Staubli VAL3: external.pjx

--- external.pjx ---
Parameters version=s7.9.4 stackSize=5000 millimeterUnit=true
Program file=aLight1.pgx
Program file=aLight2.pgx
Program file=aLight3.pgx
Program file=iCryoLongIn.pgx
Program file=iCryoShortIn.pgx
Program file=iEmergencyIn.pgx
Program file=iFluor.pgx
Program file=iFluorClosed.pgx
Program file=iFluorOpen.pgx
Program file=iGrip.pgx
Program file=iGripClosed.pgx
Program file=iGripOpen.pgx
Program file=iHeater.pgx
Program file=iIdent1.pgx
Program file=iIdent2.pgx
Program file=iIdent3.pgx
Program file=iLevel1.pgx
Program file=iLevel2.pgx
Program file=iLevel3.pgx
Program file=iLevel4.pgx
Program file=iLevel5.pgx
Program file=iLevelFault.pgx
Program file=iLidClosed.pgx
Program file=iPilatusPos.pgx
Program file=iPlate1.pgx
Program file=iPlate2.pgx
Program file=iPlate3.pgx
Program file=iPressureSensor.pgx
Program file=iRack1.pgx
Program file=iRack2.pgx
Program file=iRack3.pgx
Program file=iRack4.pgx
Program file=iSample.pgx
Program file=iSchock.pgx
Program file=iState.pgx
Program file=iTeste.pgx
Program file=iTool.pgx
Program file=ioLinks.pgx
Program file=oCryoLongOut.pgx
Program file=oCryoShortOut.pgx
Program file=oEmergencyOut.pgx
Program file=oFluorDet.pgx
Program file=oGripCmd.pgx
Program file=oGripCmd2.pgx
Program file=oHeater.pgx
Program file=oHeaterTask.pgx
Program file=oLid.pgx
Program file=oPilatusCover.pgx
Program file=oResetFault.pgx
Program file=oSample.pgx
Program file=oShutter.pgx
Program file=oVacuumValve.pgx
Program file=power.pgx
Program file=start.pgx
Program file=stop.pgx
Data file=external.dtx
Library alias=io path=io autoload=true password=

--- external.dtx ---
public aio aHeaterTime[2]
public aio aLight1[2]
public aio aLight2[2]
public aio aLight3[2]
public aio aState
public dio iCryoLongIn
public dio iCryoShortIn
public dio iEmergencyIn
public dio iFluor
public dio iFluorClosed
public dio iFluorOpen
public dio iGrip
public dio iGripClosed
public dio iGripOpen
public dio iHeaterStatus
public dio iIdent1
public dio iIdent2
public dio iIdent3
public dio iLevel1
public dio iLevel2
public dio iLevel3
public dio iLevel4
public dio iLevel5
public dio iLevelFault
public dio iLidClosed
public dio iPilatusPos
public dio iPlate1
public dio iPlate2
public dio iPlate3
public dio iPressureSensor
public dio iRack1
public dio iRack2
public dio iRack3
public dio iRack4
public dio iSampleStatus
public dio iSchock
public dio iTeste
public dio iTool
public dio oCryoLongOut
public dio oCryoShortOut
public dio oEmergencyOut
public dio oFluorDet
public dio oGripCmd
public dio oGripCmd2
public dio oHeater
public dio oLid
public dio oPilatusCover
public dio oResetFault
public dio oSample
public dio oShutter
public dio oVacuumValve
public mdesc mNomSpeed = {blend=off}

--- start.pgx ---
public program start()
begin
  call ioLinks()
end

--- aLight1.pgx ---
public program aLight1(num nValue (dimensions=1))
begin
  aioSet(aLight1,nValue)
end

--- aLight2.pgx ---
public program aLight2(num nValue (dimensions=1))
begin
  aioSet(aLight2,nValue)
end

--- aLight3.pgx ---
public program aLight3(num nValue (dimensions=1))
begin
  aioSet(aLight3,nValue)
end

--- iCryoLongIn.pgx ---
public program iCryoLongIn(num& nNum[] (dimensions=1))
begin
  nNum=dioGet(iCryoLongIn)
end

--- iCryoShortIn.pgx ---
public program iCryoShortIn(num& nNum[] (dimensions=1))
begin
  nNum=dioGet(iCryoShortIn)
end

--- iEmergencyIn.pgx ---
public program iEmergencyIn(num& nNum[] (dimensions=1))
begin
  nNum=dioGet(iEmergencyIn)
end

--- iFluor.pgx ---
public program iFluor(num& nNum[] (dimensions=1))
begin
  if (dioGet(iFluorClosed)==0) and (dioGet(iFluorOpen)==1)
    nNum=1
  endIf
  if (dioGet(iFluorClosed)==1) and (dioGet(iFluorOpen)==0)
    nNum=0
  endIf
end

--- iFluorClosed.pgx ---
public program iFluorClosed(num& nNum[] (dimensions=1))
begin
  nNum=dioGet(iFluorClosed)
end

--- iFluorOpen.pgx ---
public program iFluorOpen(num& nNum[] (dimensions=1))
begin
  nNum=dioGet(iFluorOpen)
end

--- iGrip.pgx ---
public program iGrip(num& nNum[] (dimensions=1))
begin
  if (dioGet(iGripClosed)==0) and (dioGet(iGripOpen)==1)
    nNum=1
  endIf
  if (dioGet(iGripClosed)==1) and (dioGet(iGripOpen)==0)
    nNum=0
  endIf
end

--- iGripClosed.pgx ---
public program iGripClosed(num& nNum[] (dimensions=1))
begin
  nNum=dioGet(iGripClosed)
end

--- iGripOpen.pgx ---
public program iGripOpen(num& nNum[] (dimensions=1))
begin
  nNum=dioGet(iGripOpen)
end

--- iHeater.pgx ---
public program iHeater(num& nNum[] (dimensions=1))
begin
  nNum=dioGet(iHeaterStatus)
end

--- iIdent1.pgx ---
public program iIdent1(num& nNum[] (dimensions=1))
begin
  nNum=dioGet(iIdent1)
end

--- iIdent2.pgx ---
public program iIdent2(num& nNum[] (dimensions=1))
begin
  nNum=dioGet(iIdent2)
end

--- iIdent3.pgx ---
public program iIdent3(num& nNum[] (dimensions=1))
begin
  nNum=dioGet(iIdent3)
end

--- iLevel1.pgx ---
public program iLevel1(num& nNum[] (dimensions=1))
begin
  nNum=dioGet(iLevel1)
end

--- iLevel2.pgx ---
public program iLevel2(num& nNum[] (dimensions=1))
begin
  nNum=dioGet(iLevel2)
end

--- iLevel3.pgx ---
public program iLevel3(num& nNum[] (dimensions=1))
begin
  nNum=dioGet(iLevel3)
end

--- iLevel4.pgx ---
public program iLevel4(num& nNum[] (dimensions=1))
begin
  nNum=dioGet(iLevel4)
end

--- iLevel5.pgx ---
public program iLevel5(num& nNum[] (dimensions=1))
begin
  nNum=dioGet(iLevel5)
end

--- iLevelFault.pgx ---
public program iLevelFault(num& nNum[] (dimensions=1))
begin
  nNum=dioGet(iLevelFault)
end

--- iLidClosed.pgx ---
public program iLidClosed(num& nNum[] (dimensions=1))
begin
  nNum=dioGet(iLidClosed)
end

--- ioLinks.pgx ---
program ioLinks()
begin
  dioLink(iEmergencyIn,io:EmergencyIn)
  dioLink(iSchock,io:Schock)
  dioLink(iGripOpen,io:GripOpen)
  dioLink(iGripClosed,io:GripClosed)
  dioLink(iRack1,io:Rack1)
  dioLink(iRack2,io:Rack2)
  dioLink(iRack3,io:Rack3)
  dioLink(iRack4,io:Rack4)
  dioLink(iIdent1,io:Ident1)
  dioLink(iIdent2,io:Ident2)
  dioLink(iIdent3,io:Ident3)
  dioLink(iPressureSensor,io:PressureSensor)
  dioLink(iCryoShortIn,io:CryoShortIn)
  dioLink(iCryoLongIn,io:CryoLongIn)
  dioLink(iPilatusPos,io:PilatusPos)
  dioLink(iPlate1,io:Plate1)
  dioLink(iPlate2,io:Plate2)
  dioLink(iPlate3,io:Plate3)
  dioLink(iLevelFault,io:LevelFault)
  dioLink(iLevel1,io:Level1)
  dioLink(iLevel2,io:Level2)
  dioLink(iLevel3,io:Level3)
  dioLink(iLevel4,io:Level4)
  dioLink(iLevel5,io:Level5)
  dioLink(iLidClosed,io:LidClosed)
  dioLink(iFluorOpen,io:FluorOpen)
  dioLink(iFluorClosed,io:FluorClosed)
  dioLink(iHeaterStatus,io:HeaterStatus)
  dioLink(iSampleStatus,io:SampleStatus)
  dioLink(oResetFault,io:ResetFault)
  dioLink(oEmergencyOut,io:EmergencyOut)
  dioLink(oCryoShortOut,io:CryoShortOut)
  dioLink(oCryoLongOut,io:CryoLongOut)
  dioLink(oFluorDet,io:FluorDet)
  dioLink(oPilatusCover,io:PilatusCover)
  dioLink(oLid,io:Lid)
  dioLink(oHeater,io:Heater)
  dioLink(oShutter,io:Shutter)
  dioLink(oVacuumValve,io:VacuumValve)
  dioLink(oGripCmd,io:valve1)
  dioLink(oGripCmd2,io:valve2)
  dioLink(oSample,io:Sample)
  aioLink(aLight1,io:Light1)
  aioLink(aLight2,io:Light2)
  aioLink(aLight3,io:Light3)
  aioLink(aHeaterTime,io:HeaterTime)
end

--- iPilatusPos.pgx ---
public program iPilatusPos(num& nNum[] (dimensions=1))
begin
  nNum=dioGet(iPilatusPos)
end

--- iPlate1.pgx ---
public program iPlate1(num& nNum[] (dimensions=1))
begin
  nNum=dioGet(iPlate1)
end

--- iPlate2.pgx ---
public program iPlate2(num& nNum[] (dimensions=1))
begin
  nNum=dioGet(iPlate2)
end

--- iPlate3.pgx ---
public program iPlate3(num& nNum[] (dimensions=1))
begin
  nNum=dioGet(iPlate3)
end

--- iPressureSensor.pgx ---
public program iPressureSensor(num& nNum[] (dimensions=1))
begin
  nNum=dioGet(iPressureSensor)
end

--- iRack1.pgx ---
public program iRack1(num& nNum[] (dimensions=1))
begin
  nNum=dioGet(iRack1)
end

--- iRack2.pgx ---
public program iRack2(num& nNum[] (dimensions=1))
begin
  nNum=dioGet(iRack2)
end

--- iRack3.pgx ---
public program iRack3(num& nNum[] (dimensions=1))
begin
  nNum=dioGet(iRack3)
end

--- iRack4.pgx ---
public program iRack4(num& nNum[] (dimensions=1))
begin
  nNum=dioGet(iRack4)
end

--- iSample.pgx ---
public program iSample(num& nNum[] (dimensions=1))
begin
  nNum=dioGet(iSampleStatus)
end

--- iSchock.pgx ---
public program iSchock(num& nNum[] (dimensions=1))
begin
  nNum=dioGet(iSchock)
end

--- iState.pgx ---
public program iState(num& nNum[] (dimensions=1))
begin
end

--- iTeste.pgx ---
public program iTeste(num& nNum[] (dimensions=1))
begin
end

--- iTool.pgx ---
public program iTool(num& nNum[] (dimensions=1))
begin
  nNum=dioGet(iIdent1)+(2*dioGet(iIdent2))+(4*dioGet(iIdent3))
end

--- oCryoLongOut.pgx ---
public program oCryoLongOut(num nChoice (dimensions=1))
// oCryoLongOut
begin
  dioSet(oCryoLongOut,nChoice)
end

--- oCryoShortOut.pgx ---
public program oCryoShortOut(num nChoice (dimensions=1))
// oCryoShortOut
begin
  dioSet(oCryoShortOut,nChoice)
end

--- oEmergencyOut.pgx ---
public program oEmergencyOut(num nChoice (dimensions=1))
// oEmergencyOut
begin
  dioSet(oEmergencyOut,nChoice)
end

--- oFluorDet.pgx ---
public program oFluorDet(num nChoice (dimensions=1))
// oFluorDet
begin
  dioSet(oFluorDet,nChoice)
end

--- oGripCmd.pgx ---
public program oGripCmd(num nState (dimensions=1))
begin
  dioSet(oGripCmd,nState)
end

--- oGripCmd2.pgx ---
public program oGripCmd2(num nState (dimensions=1))
begin
  dioSet(oGripCmd2,nState)
end

--- oHeater.pgx ---
public program oHeater(num nState (dimensions=1), num nDuration (dimensions=1))
begin
  switch nState
    case 0
      dioSet(oHeater,0)
      if (taskStatus("heating")==1)
        taskKill("heating")
      endIf
    break
    case 1
      taskCreate "heating",3,oHeaterTask(nDuration)
    break
    default
    break
  endSwitch
end

--- oHeaterTask.pgx ---
program oHeaterTask(num nDuration (dimensions=1))
// Heater
begin
  dioSet(oHeater,1)
  delay(nDuration)
  dioSet(oHeater,0)
end

--- oLid.pgx ---
public program oLid(num nChoice (dimensions=1))
// oLid
begin
  dioSet(oLid,nChoice)
end

--- oPilatusCover.pgx ---
public program oPilatusCover(num nChoice (dimensions=1))
// oPilatusCover
begin
  dioSet(oPilatusCover,nChoice)
end

--- oResetFault.pgx ---
public program oResetFault()
// Reseta rele de seguranca
begin
  dioSet(oResetFault,1)
  delay(1)
  dioSet(oResetFault,0)
end

--- oSample.pgx ---
public program oSample(num nChoice (dimensions=1))
// oSample
begin
  dioSet(oSample,nChoice)
end

--- oShutter.pgx ---
public program oShutter(num nChoice (dimensions=1))
// oShutter
begin
  dioSet(oShutter,nChoice)
end

--- oVacuumValve.pgx ---
public program oVacuumValve(num nChoice (dimensions=1))
// oVacuumValve
begin
  dioSet(oVacuumValve,nChoice)
end

--- power.pgx ---
public program power(bool bState (dimensions=1), bool& bFlag[] (dimensions=1))
begin
  switch bState
    case false
      disablePower()
      bFlag=true
    break
    case true
      enablePower()
      if (watch(isPowered(),3)==false)
        bFlag=false
      else
        bFlag=true
      endIf
    break
  endSwitch
end
